TYPE
    ST_CylinderMonitor :
    STRUCT
        InFrontPosition : BOOL;
        InRearPosition  : BOOL;
        Error           : BOOL;
        ErrMsg          : T_MaxString;
    END_STRUCT
END_TYPE

(* stored: Version 1.1.0.1, ProductVersion 3.1.4024.13
   DUT ST_CylinderMonitor: Id {4d780b7a-197c-47a5-8233-646e1e334248} *)
